// TIA Portal project "Practico_8_desplazamientoPorCinta" (V15)

(* hardware
DEVICE "S7-1200 station_1"  S7-1200 Station
   slot 0: "Rack_0"  S7-1200 Rack  Rack  V1.0
   slot 1: "PLC_1"  CPU 1214C AC/DC/Rly  6ES7 214-1BG40-0XB0  V4.2
   slot 3: "AQ 1x12BIT_1"  AQ1 signal board  6ES7 232-4HA30-0XB0  V1.0
DEVICE "HMI_1"  KTP700 Basic PN
   slot 0: "HMI_1"  KTP700 Basic PN  6AV2 123-2GB03-0AX0  15.0.0.0
   slot 1: "HMI_RT_1"  KTP700 Basic PN  6AV2 123-2GB03-0AX0  15.0.0.0
   slot 5: "HMI_1.IE_CP_1"  PROFINET Interface  15.0.0.0
      slot 1: "Interfaz PROFINET_1"  PROFINET Interface
         slot 1: "Port_1"  Port
*)

// ===== PLC "PLC_1"  CPU 1214C AC/DC/Rly =====

VAR_GLOBAL   // PLC tag table "Tabla de variables estándar"
   "arriba" AT %M5.0 : Bool;
   "abajo" AT %M5.1 : Bool;
   "izquierda" AT %M5.2 : Bool;
   "derecha" AT %M5.3 : Bool;
   "PM" AT %M7.0 : Bool;
   "grua a la izquierda" AT %Q0.0 : Bool;
   "grua a la derecha" AT %Q0.1 : Bool;
   "grua arriba" AT %Q0.2 : Bool;
   "grua abajo" AT %Q0.3 : Bool;
   "Paro" AT %M7.1 : Bool;
   "bucle" AT %M5.4 : Bool;
   "System_Byte" AT %MB254 : Byte;
   "FirstScan" AT %M254.0 : Bool;
   "DiagStatusUpdate" AT %M254.1 : Bool;
   "AlwaysTRUE" AT %M254.2 : Bool;
   "AlwaysFALSE" AT %M254.3 : Bool;
   "Clock_Byte" AT %MB255 : Byte;
   "Clock_10Hz" AT %M255.0 : Bool;
   "Clock_5Hz" AT %M255.1 : Bool;
   "Clock_2.5Hz" AT %M255.2 : Bool;
   "Clock_2Hz" AT %M255.3 : Bool;
   "Clock_1.25Hz" AT %M255.4 : Bool;
   "Clock_1Hz" AT %M255.5 : Bool;
   "Clock_0.625Hz" AT %M255.6 : Bool;
   "Clock_0.5Hz" AT %M255.7 : Bool;
   "conteo" AT %MW10 : Int;
   "conteo 2" AT %MW12 : Int;
   "subiendo" AT %M5.5 : Bool;
   "hacia la izquierda" AT %M5.6 : Bool;
   "Tag_1" AT %M5.7 : Bool;
   "Tag_2" AT %M6.0 : Bool;
   "Tag_3" AT %M6.1 : Bool;
END_VAR

// folder: System blocks/Program resources

DATA_BLOCK "IEC_Counter_0_DB"   // DB1
{ S7_Optimized_Access := 'TRUE' }
AUTHOR : Simatic
FAMILY : IEC
NAME : CNTR
VERSION : 1.0
// stored: InstanceOfName IEC_COUNTER
"IEC_COUNTER"
BEGIN
END_DATA_BLOCK

DATA_BLOCK "IEC_Counter_0_DB_1"   // DB2
{ S7_Optimized_Access := 'TRUE' }
AUTHOR : Simatic
FAMILY : IEC
NAME : CNTR
VERSION : 1.0
// stored: InstanceOfName IEC_COUNTER
"IEC_COUNTER"
BEGIN
END_DATA_BLOCK

DATA_BLOCK "IEC_Timer_0_DB"   // DB3
{ S7_Optimized_Access := 'TRUE' }
AUTHOR : Simatic
FAMILY : IEC
NAME : IEC_TMR
VERSION : 1.0
// stored: InstanceOfName IEC_TIMER
"IEC_TIMER"
BEGIN
END_DATA_BLOCK

DATA_BLOCK "IEC_Timer_0_DB_1"   // DB4
{ S7_Optimized_Access := 'TRUE' }
AUTHOR : Simatic
FAMILY : IEC
NAME : IEC_TMR
VERSION : 1.0
// stored: InstanceOfName IEC_TIMER
"IEC_TIMER"
BEGIN
END_DATA_BLOCK

// folder: (top level)

ORGANIZATION_BLOCK "Main"   // OB1, LAD, ProgramCycle
TITLE = "Main Program Sweep (Cycle)"
{ S7_Optimized_Access := 'TRUE' }
VERSION : 0.1
   VAR_INPUT
      Initial_Call : Bool;   // Initial call of this OB
      Remanence : Bool;   // =True, if remanent data are available
   END_VAR
   VAR_TEMP   // added for the SCL form of the ladder/FBD networks
      _w1 : Bool;
      _w2 : Bool;
      _w3 : Bool;
      _w4 : Bool;
   END_VAR
BEGIN

REGION Network 1: Marcha
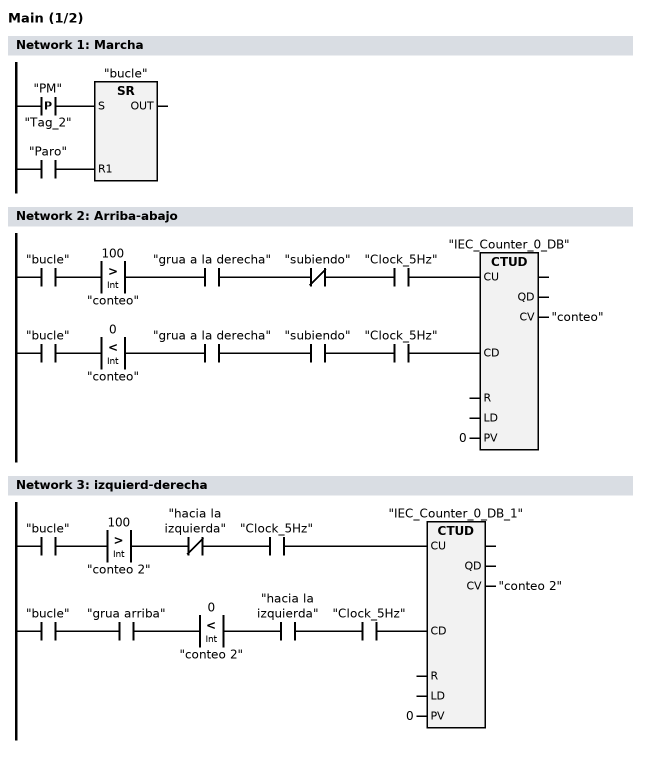
   RUNG wire#powerrail
      P_Contact(operand := "PM", bit := "Tag_2")
      S_SR(operand := "bucle", r1 := wire#w1)
   END_RUNG
   RUNG wire#powerrail
      Contact( "Paro" )
   END_RUNG wire#w1
   // the same network as SCL:
   #_w1 := "PM" AND NOT "Tag_2";   // rising edge of "PM"
   "Tag_2" := "PM";
   IF #_w1 THEN
       "bucle" := TRUE;   // SR flip-flop
   END_IF;
   IF "Paro" THEN "bucle" := FALSE; END_IF;
END_REGION

REGION Network 2: Arriba-abajo
   "IEC_Counter_0_DB".CTUD(CU := "bucle" AND (100 > "conteo") AND "grua a la derecha" AND NOT "subiendo" AND "Clock_5Hz",
                           CD := "bucle" AND (0 < "conteo") AND "grua a la derecha" AND "subiendo" AND "Clock_5Hz",
                           PV := 0,
                           CV => "conteo");
END_REGION

REGION Network 3: izquierd-derecha
   "IEC_Counter_0_DB_1".CTUD(CU := "bucle" AND (100 > "conteo 2") AND NOT "hacia la izquierda" AND "Clock_5Hz",
                           CD := "bucle" AND "grua arriba" AND (0 < "conteo 2") AND "hacia la izquierda" AND "Clock_5Hz",
                           PV := 0,
                           CV => "conteo 2");
END_REGION

REGION Network 4: Finales de carrera
   // el conteo uno se refiere al proceso de subir y bajar y el conteo 2 al proceso de ir a la izquierda o derecha.
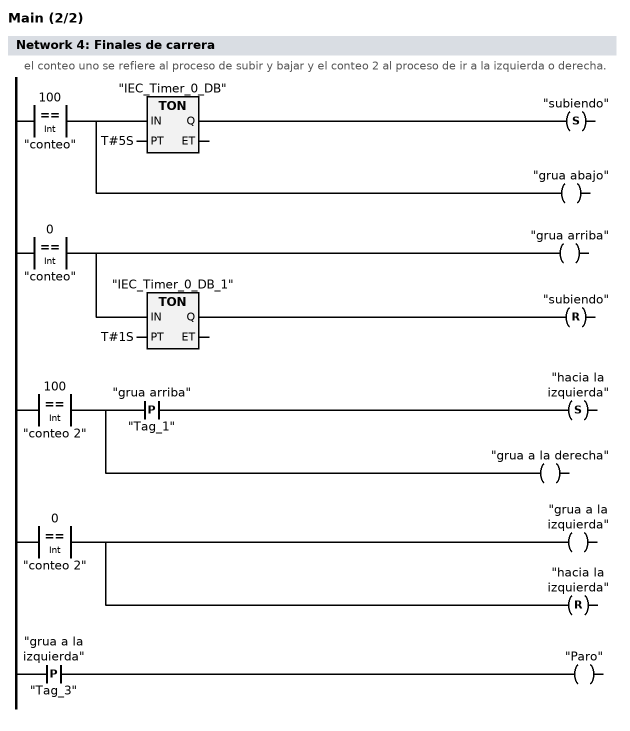
   #_w1 := 100 = "conteo";
   "IEC_Timer_0_DB".TON(IN := #_w1, PT := T#5S);
   IF "IEC_Timer_0_DB".Q THEN "subiendo" := TRUE; END_IF;
   "grua abajo" := #_w1;
   "grua arriba" := 0 = "conteo";
   "IEC_Timer_0_DB_1".TON(IN := "grua arriba", PT := T#1S);
   IF "IEC_Timer_0_DB_1".Q THEN "subiendo" := FALSE; END_IF;
   #_w2 := 100 = "conteo 2";
   #_w3 := #_w2 AND "grua arriba" AND NOT "Tag_1";   // rising edge of "grua arriba"
   "Tag_1" := "grua arriba";
   IF #_w3 THEN "hacia la izquierda" := TRUE; END_IF;
   "grua a la derecha" := #_w2;
   "grua a la izquierda" := 0 = "conteo 2";
   IF "grua a la izquierda" THEN "hacia la izquierda" := FALSE; END_IF;
   #_w4 := "grua a la izquierda" AND NOT "Tag_3";   // rising edge of "grua a la izquierda"
   "Tag_3" := "grua a la izquierda";
   "Paro" := #_w4;
END_REGION
END_ORGANIZATION_BLOCK

(* ===== HMI "HMI_RT_1" =====
system functions are stored by id; their names below are inferred from use
connection "HMI_Conexión_1": ETHERNET, SMART_S7_1200_OMS

HMI tags "Tabla de variables estándar"
   "Número_imagen_variable" : UInt, internal
   "conteo 2" : Int = PLC "conteo 2" AT %MW12, 1 s
   "conteo" : Int = PLC conteo AT %MW10, 1 s
   "PM" : Bool = PLC PM AT %M7.0, 1 s
   "Paro" : Bool = PLC Paro AT %M7.1, 1 s
   "grua a la derecha" : Bool = PLC "grua a la derecha" AT %Q0.1, 1 s

text list "Nombre_imagen_lista_texto": 1 'Imagen raíz'

Template "Plantilla_1" 800x480
   Button "Salir" at 714,429 size 71x50; TextOff 'Salir'; PictureOff "ExitRuntime_KTP700_Basic_PN_TR"; PictureOn "ExitRuntime_KTP700_Basic_PN_TR"
      on Release: StopRuntime(0)
   Button "Template_Button" at 614,429 size 71x50; TextOff 'Text'
   Button "Template_Button_1" at 514,429 size 71x50; TextOff 'Text'
   Button "Template_Button_2" at 414,429 size 71x50; TextOff 'Text'
   Button "Template_Button_3" at 314,429 size 71x50; TextOff 'Text'
   Button "Template_Button_4" at 214,429 size 71x50; TextOff 'Text'
   Button "Avisos" at 114,429 size 71x50; TextOff 'Avisos'; PictureOff "AlarmDisplay_KTP700_Basic_PN_TR"; PictureOn "AlarmDisplay_KTP700_Basic_PN_TR"
      on Release: function_ef3f5d25("Ventana de avisos_no_acusado", -1)
   Button "Imagen inicial" at 14,429 size 71x50; TextOff 'Imagen inicial'; PictureOff "NavigateHome_KTP700_Basic_PN_TR"; PictureOn "NavigateHome_KTP700_Basic_PN_TR"
      on Release: ActivateScreen("Imagen raíz", 0)
   SymbolicIOField "Imagen_campo_ES_simbólico" at 93,9 size 600x33; TextOff '0'; TextOn '1'; TextList "Nombre_imagen_lista_texto"
      ProcessValue <- "Número_imagen_variable"
      on Change: ActivateScreenByNumber("Número_imagen_variable", 0)
   DateTimeField "HmiScreenItemData" at 695,25 size 105x25
   DateTimeField "HmiScreenItemData_1" at 695,0 size 105x25
   GraphicView "Logotipo" at 0,0 size 91x51; Picture "Logotipo de HMI_1"

screen "Imagen raíz" 800x480, template "Plantilla_1"
   on GenerateScreen: SetTag("Número_imagen_variable", 1)
   Button "Botón_1" at 600,182 size 96x32; TextOff 'PM'
      on Press: SetBit("PM")
      on Release: ResetBit("PM")
   Button "Botón_2" at 601,239 size 96x32; TextOff 'Paro'
      on Press: SetBit("Paro")
      on Release: ResetBit("Paro")
   GraphicView "Visor de gráficos_3" at 73,76 size 560x48; Picture "grua_2"
   GraphicView "Visor de gráficos_1" at 121,119 size 36x46; Picture "kisspng-hook-vector-graphics-crane-metal-excavator-5c03144b3c6c67.1317103015437056752475"
      HorizontalMovement <- "conteo 2"
      Visibility <- "conteo 2"
   GraphicView "Visor de gráficos_2" at 520,120 size 36x45; Picture "kisspng-hook-vector-graphics-crane-metal-excavator-5c03144b3c6c67.1317103015437056752475"
      VerticalMovement <- "conteo"
      Visibility <- "conteo 2"
*)